SUBAPPLICATION Uebung_012e2_AR (* Numeric Value Input PHYS und Speichern INI mit Subapp (AR Adapter) *)
  (* Standard: 61499-2; Description: Copyright (c) 2026 Meisterschulen am Ostbahnhof This program and the accompanying materials are made available under the terms of the Eclipse Public License 2.0 which is available at https://www.eclipse.org/legal/epl-2.0/ SPDX-License-Identifier: EPL-2.0 *)
  (* Version 1.0, 2026-04-24, Franz Höpfinger, Meisterschulen am Ostbahnhof, AR adapter variant of Uebung_012e *)
  PACKAGE Uebungen;
  IMPORT Uebungen::const::NVS::NVS_Keys::KEY_I1_STORE;
  IMPORT Uebungen::const::NVS::NVS_Keys::SECTION_I1_STORE;
  IMPORT logiBUS::io::DI::logiBUS_DI::Input_I1;
  IMPORT logiBUS::io::DQ::logiBUS_DO::Output_Q1;
  IMPORT Uebungen::const::UT::DefaultPool_Numeric::InputNumber_I3_N;
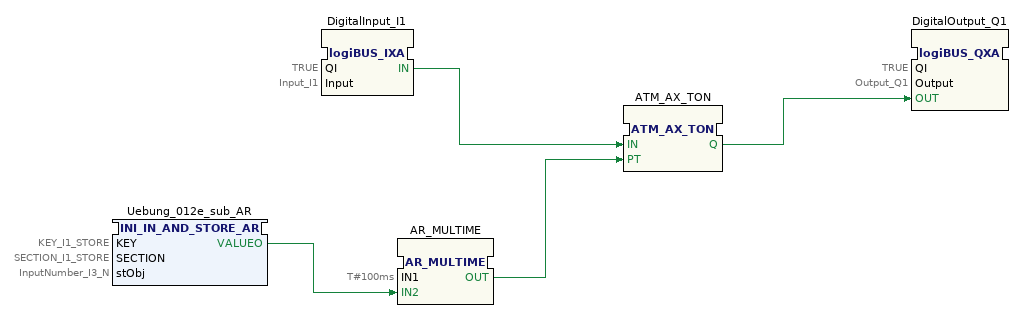
  (* Einstellbarer Timer *)
  FBS
    DigitalOutput_Q1 : logiBUS::io::DQ::logiBUS_QXA(QI := TRUE, Output := Output_Q1);
    ATM_AX_TON : adapter::events::unidirectional::timers::ATM_AX_TON;
    DigitalInput_I1 : logiBUS::io::DI::logiBUS_IXA(QI := TRUE, Input := Input_I1);
    AR_MULTIME : adapter::iec61131::arithmetic::AR_MULTIME(IN1 := T#100ms);
  END_FBS
  SUBAPPS
    Uebung_012e_sub_AR : MyLib::sys::INI_IN_AND_STORE_AR(KEY := KEY_I1_STORE, SECTION := SECTION_I1_STORE, stObj := InputNumber_I3_N);
  END_SUBAPPS
  ADAPTER_CONNECTIONS
    DigitalInput_I1.IN TO ATM_AX_TON.IN;
    ATM_AX_TON.Q TO DigitalOutput_Q1.OUT;
    Uebung_012e_sub_AR.VALUEO TO AR_MULTIME.IN2;
    AR_MULTIME.OUT TO ATM_AX_TON.PT;
  END_CONNECTIONS
END_SUBAPPLICATION
